# EPICS StreamDevice protocol: tjmperSup/tjmper.proto
Terminator = CR;
ReplyTimeout = 1000;

getStatus {
    out "?STS";
    in "ACK";
    in "ITJ%d,OPM%(\$1MODE)d,LMT%(\$1LMT)d,AIR%(\$1AIR)d,ERR%(\$1ERR)d";
}

setMode {
    out "%{OPM0|OPM1|OPM2}";
    in "ACK";
}
